// TIA Portal V20 export
// export: Created 2026-07-16T12:59:01.3797078Z, ExportSetting WithDefaults, DisplayName Totally Integrated Automation Portal, DisplayVersion V20 Update 5, DisplayName TIA Portal Openness, DisplayVersion V20 Update 4, DisplayName TIA Portal Version Control Interface, DisplayVersion V20 Update 5, DisplayName SINAMICS Startdrive Advanced, DisplayVersion V20, DisplayName SINAMICS DCC, DisplayVersion V20, DisplayName SINAMICS Startdrive G130, G150, S120, S150, SINAMICS MV, G220, S200, S210, DisplayVersion V20, DisplayName SINAMICS Startdrive G110M, G120, G120C, G120D, G120P, G115D, DisplayVersion V20, DisplayName STEP 7 Professional, DisplayVersion V20 Update 5, DisplayName STEP 7 Safety, DisplayVersion V20 Update 2, DisplayName WinCC Basic/Comfort/Advanced, DisplayVersion V20 Update 5, DisplayName WinCC Unified, DisplayVersion V20 Update 5
FUNCTION_BLOCK "FB_MotorFwdRevSystem"   // FB7, LAD
{ S7_Optimized_Access := 'TRUE' }
VERSION : 0.1
// stored: AutoNumber true, IsIECCheckEnabled false, IsRetainMemResEnabled false, MemoryReserve 100, SetENOAutomatically false, UDAEnableTagReadback false
   VAR RETAIN
      IO : "MotorFwdRevIOSet";
   END_VAR
   VAR
      RisingEdgeFlags : Array[0..3] of Bool;
      NegitiveSignalEdge : Array[0..2] of Bool;
      Pasue : Bool;
      HrTotaliserTimerReset : Bool;
      EnableUPSTimeMS : DInt;
      ShutdownTimeMS : DInt;
      FTTimeMS : DInt;
      PauseTimeMS : DInt;
      ReverseIgnoreFTTimeMS : DInt;
      FaultTripTimer { S7_SetPoint := 'True'} : TON_TIME;
      FTSTimer { S7_SetPoint := 'True'} : TON_TIME;
      EnableUpstreamTimer { S7_SetPoint := 'True'} : TON_TIME;
      ShutdownTimer { S7_SetPoint := 'True'} : TON_TIME;
      GeneralDelayTimer { S7_SetPoint := 'True'} : TON_TIME;
      InHandReqPreStart { S7_SetPoint := 'True'} : TON_TIME;
      CycleDelayReset { S7_SetPoint := 'True'} : TON_TIME;
   END_VAR
   VAR RETAIN
      HrTotaliserTimer { S7_SetPoint := 'True'} : TONR_TIME;
   END_VAR
   VAR
      ReversalPauseTimer { S7_SetPoint := 'True'} : TON_TIME;
      ReversalIgnoreFTTimer { S7_SetPoint := 'True'} : TON_TIME;
      PreStartMemory { S7_SetPoint := 'True'} : Bool;
      HandPosEdge : Bool;
      HandNegEdge : Bool;
      CycleDelay : Bool;
   END_VAR
   VAR_TEMP
      "Time" : Real;
      StartTimer : Bool;
   END_VAR
   VAR_TEMP   // added for the SCL form of the ladder/FBD networks
      _w1 : Bool;
      _w2 : Bool;
   END_VAR
BEGIN

REGION Network 1: Reverse Pause and Control
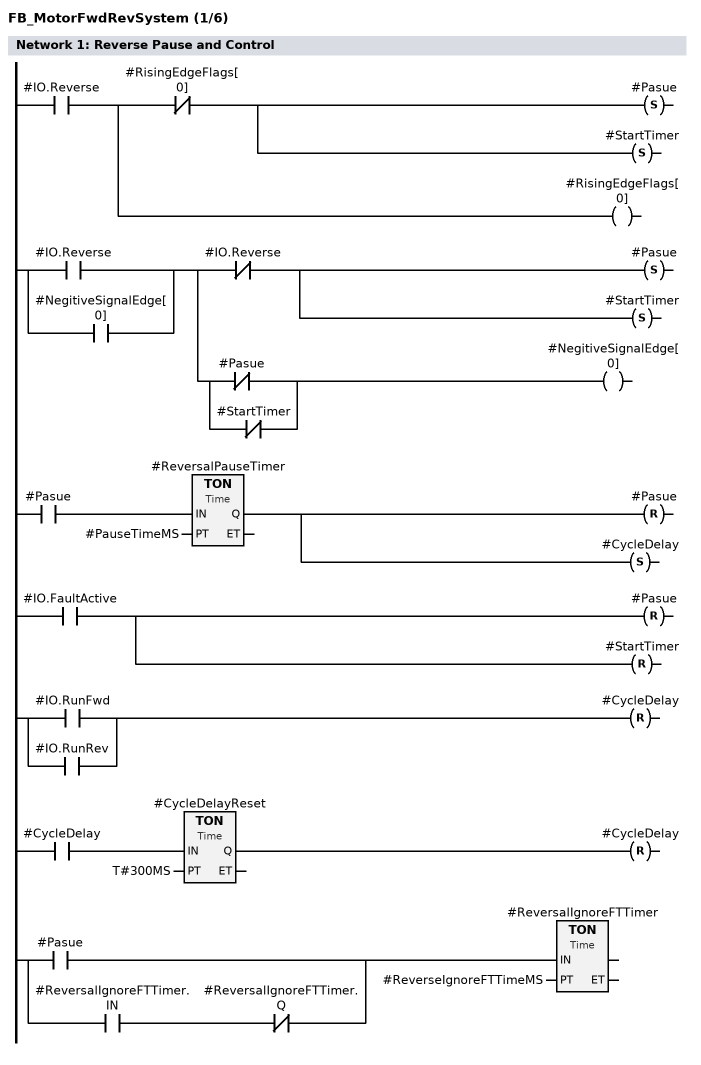
   RUNG wire#powerrail
      Contact( #IO.Reverse )
      wire#w1
      I_Contact( #RisingEdgeFlags[0] )
      wire#w2
      S_Coil( #Pasue )
   END_RUNG
   RUNG wire#w2
      S_Coil( #StartTimer )
   END_RUNG
   RUNG wire#w1
      Coil( #RisingEdgeFlags[0] )
   END_RUNG
   RUNG wire#powerrail
      Contact( #IO.Reverse )
      wire#w3
      I_Contact( #IO.Reverse )
      wire#w4
      S_Coil( #Pasue )
   END_RUNG
   RUNG wire#powerrail
      Contact( #NegitiveSignalEdge[0] )
   END_RUNG wire#w3
   RUNG wire#w4
      S_Coil( #StartTimer )
   END_RUNG
   RUNG wire#w3
      I_Contact( #Pasue )
      wire#w5
      Coil( #NegitiveSignalEdge[0] )
   END_RUNG
   RUNG wire#w3
      I_Contact( #StartTimer )
   END_RUNG wire#w5
   RUNG wire#powerrail
      Contact( #Pasue )
      { S7_Templates := "time_type := Time" } #ReversalPauseTimer.TON(pt := #PauseTimeMS, et =>)
      wire#w6
      R_Coil( #Pasue )
   END_RUNG
   RUNG wire#w6
      S_Coil( #CycleDelay )
   END_RUNG
   RUNG wire#powerrail
      Contact( #IO.FaultActive )
      wire#w7
      R_Coil( #Pasue )
   END_RUNG
   RUNG wire#w7
      R_Coil( #StartTimer )
   END_RUNG
   RUNG wire#powerrail
      Contact( #IO.RunFwd )
      wire#w8
      R_Coil( #CycleDelay )
   END_RUNG
   RUNG wire#powerrail
      Contact( #IO.RunRev )
   END_RUNG wire#w8
   RUNG wire#powerrail
      Contact( #CycleDelay )
      { S7_Templates := "time_type := Time" } #CycleDelayReset.TON(pt := T#300MS, et =>)
      R_Coil( #CycleDelay )
   END_RUNG
   RUNG wire#powerrail
      Contact( #Pasue )
      wire#w9
      { S7_Templates := "time_type := Time" } #ReversalIgnoreFTTimer.TON(pt := #ReverseIgnoreFTTimeMS, et =>)
   END_RUNG
   RUNG wire#powerrail
      Contact( #ReversalIgnoreFTTimer.IN )
      I_Contact( #ReversalIgnoreFTTimer.Q )
   END_RUNG wire#w9
   // the same network as SCL:
   IF #IO.Reverse AND NOT #RisingEdgeFlags[0] THEN
       #Pasue := TRUE;
       #StartTimer := TRUE;
   END_IF;
   #RisingEdgeFlags[0] := #IO.Reverse;
   #_w1 := #IO.Reverse OR #NegitiveSignalEdge[0];
   IF #_w1 AND NOT #IO.Reverse THEN
       #Pasue := TRUE;
       #StartTimer := TRUE;
   END_IF;
   #NegitiveSignalEdge[0] := #_w1 AND (NOT #Pasue OR NOT #StartTimer);
   #ReversalPauseTimer(IN := #Pasue, PT := #PauseTimeMS);   // TON
   IF #ReversalPauseTimer.Q THEN
       #Pasue := FALSE;
       #CycleDelay := TRUE;
   END_IF;
   IF #IO.FaultActive THEN
       #Pasue := FALSE;
       #StartTimer := FALSE;
   END_IF;
   IF #IO.RunFwd OR #IO.RunRev THEN #CycleDelay := FALSE; END_IF;
   #CycleDelayReset(IN := #CycleDelay, PT := T#300MS);   // TON
   IF #CycleDelayReset.Q THEN #CycleDelay := FALSE; END_IF;
   #ReversalIgnoreFTTimer(IN := #Pasue OR (#ReversalIgnoreFTTimer.IN AND NOT #ReversalIgnoreFTTimer.Q),   // TON
                          PT := #ReverseIgnoreFTTimeMS);
END_REGION

REGION Network 2: DOL Motor Start / Stop
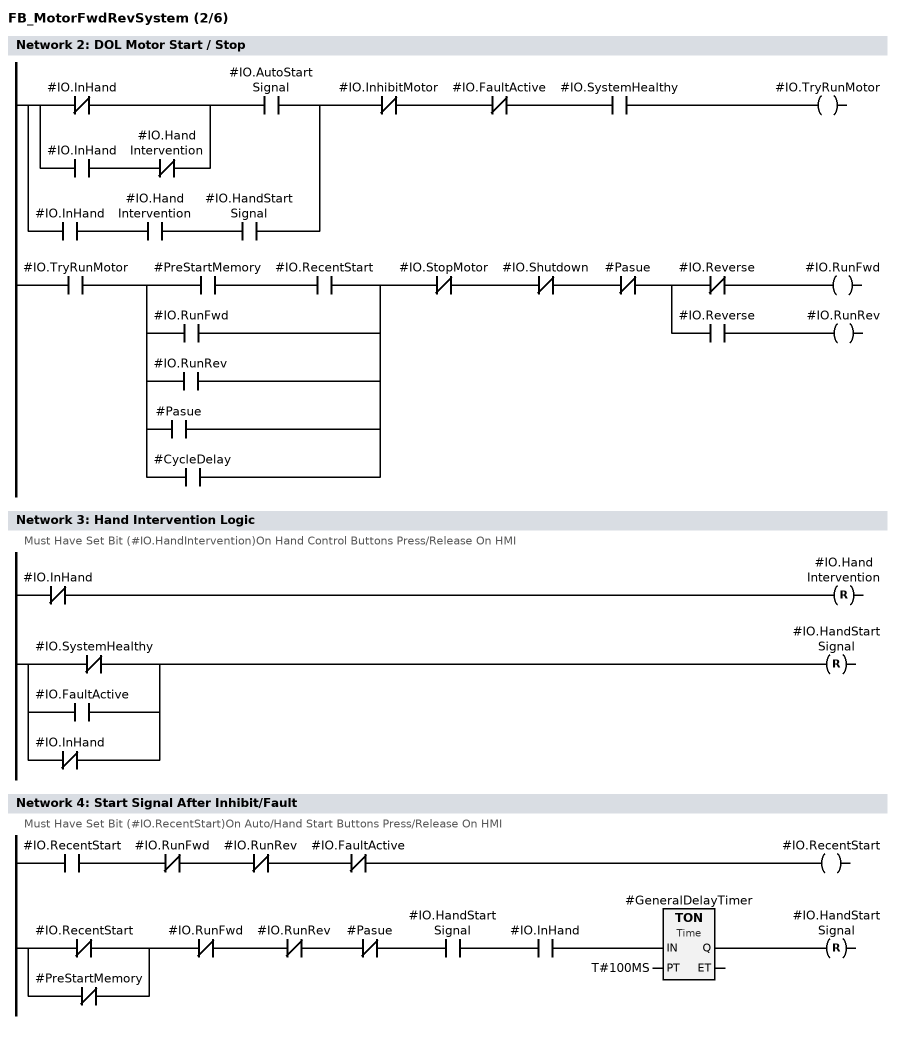
   RUNG wire#powerrail
      I_Contact( #IO.InHand )
      wire#w1
      Contact( #IO.AutoStartSignal )
      wire#w2
      I_Contact( #IO.InhibitMotor )
      I_Contact( #IO.FaultActive )
      Contact( #IO.SystemHealthy )
      Coil( #IO.TryRunMotor )
   END_RUNG
   RUNG wire#powerrail
      Contact( #IO.InHand )
      I_Contact( #IO.HandIntervention )
   END_RUNG wire#w1
   RUNG wire#powerrail
      Contact( #IO.InHand )
      Contact( #IO.HandIntervention )
      Contact( #IO.HandStartSignal )
   END_RUNG wire#w2
   RUNG wire#powerrail
      Contact( #IO.TryRunMotor )
      wire#w3
      Contact( #PreStartMemory )
      Contact( #IO.RecentStart )
      wire#w4
      I_Contact( #IO.StopMotor )
      I_Contact( #IO.Shutdown )
      I_Contact( #Pasue )
      wire#w5
      I_Contact( #IO.Reverse )
      Coil( #IO.RunFwd )
   END_RUNG
   RUNG wire#w3
      Contact( #IO.RunFwd )
   END_RUNG wire#w4
   RUNG wire#w3
      Contact( #IO.RunRev )
   END_RUNG wire#w4
   RUNG wire#w3
      Contact( #Pasue )
   END_RUNG wire#w4
   RUNG wire#w3
      Contact( #CycleDelay )
   END_RUNG wire#w4
   RUNG wire#w5
      Contact( #IO.Reverse )
      Coil( #IO.RunRev )
   END_RUNG
   // the same network as SCL:
   #IO.TryRunMotor := (((NOT #IO.InHand OR (#IO.InHand AND NOT #IO.HandIntervention)) AND #IO.AutoStartSignal) OR (#IO.InHand AND #IO.HandIntervention AND #IO.HandStartSignal)) AND NOT #IO.InhibitMotor AND NOT #IO.FaultActive AND #IO.SystemHealthy;
   #_w1 := #IO.TryRunMotor AND ((#PreStartMemory AND #IO.RecentStart) OR #IO.RunFwd OR #IO.RunRev OR #Pasue OR #CycleDelay) AND NOT #IO.StopMotor AND NOT #IO.Shutdown AND NOT #Pasue;
   #IO.RunFwd := #_w1 AND NOT #IO.Reverse;
   #IO.RunRev := #_w1 AND #IO.Reverse;
END_REGION

REGION Network 3: Hand Intervention Logic
   // Must Have Set Bit (#IO.HandIntervention)On Hand Control Buttons Press/Release On HMI
   RUNG wire#powerrail
      I_Contact( #IO.InHand )
      R_Coil( #IO.HandIntervention )
   END_RUNG
   RUNG wire#powerrail
      I_Contact( #IO.SystemHealthy )
      wire#w1
      R_Coil( #IO.HandStartSignal )
   END_RUNG
   RUNG wire#powerrail
      Contact( #IO.FaultActive )
   END_RUNG wire#w1
   RUNG wire#powerrail
      I_Contact( #IO.InHand )
   END_RUNG wire#w1
   // the same network as SCL:
   IF NOT #IO.InHand THEN #IO.HandIntervention := FALSE; END_IF;
   IF NOT #IO.SystemHealthy OR #IO.FaultActive OR NOT #IO.InHand THEN #IO.HandStartSignal := FALSE; END_IF;
END_REGION

REGION Network 4: Start Signal After Inhibit/Fault
   // Must Have Set Bit (#IO.RecentStart)On Auto/Hand Start Buttons Press/Release On HMI
   RUNG wire#powerrail
      Contact( #IO.RecentStart )
      I_Contact( #IO.RunFwd )
      I_Contact( #IO.RunRev )
      I_Contact( #IO.FaultActive )
      Coil( #IO.RecentStart )
   END_RUNG
   RUNG wire#powerrail
      I_Contact( #IO.RecentStart )
      wire#w1
      I_Contact( #IO.RunFwd )
      I_Contact( #IO.RunRev )
      I_Contact( #Pasue )
      Contact( #IO.HandStartSignal )
      Contact( #IO.InHand )
      { S7_Templates := "time_type := Time" } #GeneralDelayTimer.TON(pt := T#100MS, et =>)
      R_Coil( #IO.HandStartSignal )
   END_RUNG
   RUNG wire#powerrail
      I_Contact( #PreStartMemory )
   END_RUNG wire#w1
   // the same network as SCL:
   #IO.RecentStart := #IO.RecentStart AND NOT #IO.RunFwd AND NOT #IO.RunRev AND NOT #IO.FaultActive;
   #GeneralDelayTimer(IN := (NOT #IO.RecentStart OR NOT #PreStartMemory) AND NOT #IO.RunFwd AND NOT #IO.RunRev AND NOT #Pasue AND #IO.HandStartSignal AND #IO.InHand,   // TON
                      PT := T#100MS);
   IF #GeneralDelayTimer.Q THEN #IO.HandStartSignal := FALSE; END_IF;
END_REGION

REGION Network 5
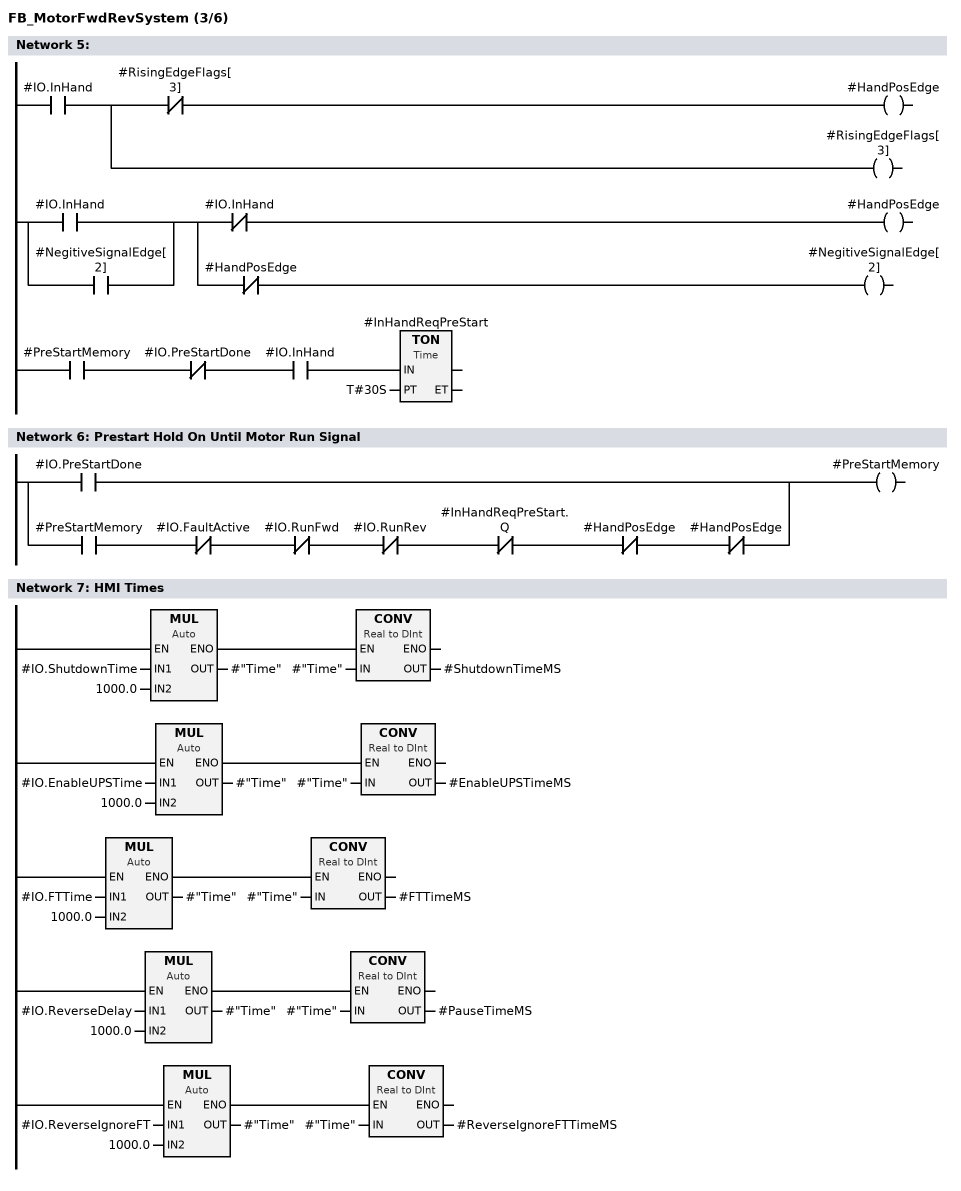
   RUNG wire#powerrail
      Contact( #IO.InHand )
      wire#w1
      I_Contact( #RisingEdgeFlags[3] )
      Coil( #HandPosEdge )
   END_RUNG
   RUNG wire#w1
      Coil( #RisingEdgeFlags[3] )
   END_RUNG
   RUNG wire#powerrail
      Contact( #IO.InHand )
      wire#w2
      I_Contact( #IO.InHand )
      Coil( #HandPosEdge )
   END_RUNG
   RUNG wire#powerrail
      Contact( #NegitiveSignalEdge[2] )
   END_RUNG wire#w2
   RUNG wire#w2
      I_Contact( #HandPosEdge )
      Coil( #NegitiveSignalEdge[2] )
   END_RUNG
   RUNG wire#powerrail
      Contact( #PreStartMemory )
      I_Contact( #IO.PreStartDone )
      Contact( #IO.InHand )
      { S7_Templates := "time_type := Time" } #InHandReqPreStart.TON(pt := T#30S, et =>)
   END_RUNG
   // the same network as SCL:
   #HandPosEdge := #IO.InHand AND NOT #RisingEdgeFlags[3];
   #RisingEdgeFlags[3] := #IO.InHand;
   #_w1 := #IO.InHand OR #NegitiveSignalEdge[2];
   #HandPosEdge := #_w1 AND NOT #IO.InHand;
   #NegitiveSignalEdge[2] := #_w1 AND NOT #HandPosEdge;
   #InHandReqPreStart(IN := #PreStartMemory AND NOT #IO.PreStartDone AND #IO.InHand, PT := T#30S);   // TON
END_REGION

REGION Network 6: Prestart Hold On Until Motor Run Signal
   RUNG wire#powerrail
      Contact( #IO.PreStartDone )
      wire#w1
      Coil( #PreStartMemory )
   END_RUNG
   RUNG wire#powerrail
      Contact( #PreStartMemory )
      I_Contact( #IO.FaultActive )
      I_Contact( #IO.RunFwd )
      I_Contact( #IO.RunRev )
      I_Contact( #InHandReqPreStart.Q )
      I_Contact( #HandPosEdge )
      I_Contact( #HandPosEdge )
   END_RUNG wire#w1
   // the same network as SCL:
   #PreStartMemory := #IO.PreStartDone OR (#PreStartMemory AND NOT #IO.FaultActive AND NOT #IO.RunFwd AND NOT #IO.RunRev AND NOT #InHandReqPreStart.Q AND NOT #HandPosEdge AND NOT #HandPosEdge);
END_REGION

REGION Network 7: HMI Times
   RUNG wire#powerrail
      Mul(in1 := #IO.ShutdownTime, in2 := 1000.0, out => #"Time")
      { S7_Templates := "[SrcType := Real, DestType := DInt]" } Convert(in := #"Time", out => #ShutdownTimeMS)
   END_RUNG
   RUNG wire#powerrail
      Mul(in1 := #IO.EnableUPSTime, in2 := 1000.0, out => #"Time")
      { S7_Templates := "[SrcType := Real, DestType := DInt]" } Convert(in := #"Time", out => #EnableUPSTimeMS)
   END_RUNG
   RUNG wire#powerrail
      Mul(in1 := #IO.FTTime, in2 := 1000.0, out => #"Time")
      { S7_Templates := "[SrcType := Real, DestType := DInt]" } Convert(in := #"Time", out => #FTTimeMS)
   END_RUNG
   RUNG wire#powerrail
      Mul(in1 := #IO.ReverseDelay, in2 := 1000.0, out => #"Time")
      { S7_Templates := "[SrcType := Real, DestType := DInt]" } Convert(in := #"Time", out => #PauseTimeMS)
   END_RUNG
   RUNG wire#powerrail
      Mul(in1 := #IO.ReverseIgnoreFT, in2 := 1000.0, out => #"Time")
      { S7_Templates := "[SrcType := Real, DestType := DInt]" } Convert(in := #"Time", out => #ReverseIgnoreFTTimeMS)
   END_RUNG
   // the same network as SCL:
   #"Time" := #IO.ShutdownTime * 1000.0;
   #ShutdownTimeMS := REAL_TO_DINT(#"Time");
   #"Time" := #IO.EnableUPSTime * 1000.0;
   #EnableUPSTimeMS := REAL_TO_DINT(#"Time");
   #"Time" := #IO.FTTime * 1000.0;
   #FTTimeMS := REAL_TO_DINT(#"Time");
   #"Time" := #IO.ReverseDelay * 1000.0;
   #PauseTimeMS := REAL_TO_DINT(#"Time");
   #"Time" := #IO.ReverseIgnoreFT * 1000.0;
   #ReverseIgnoreFTTimeMS := REAL_TO_DINT(#"Time");
END_REGION

REGION Network 8: DOL Motor Shutdown
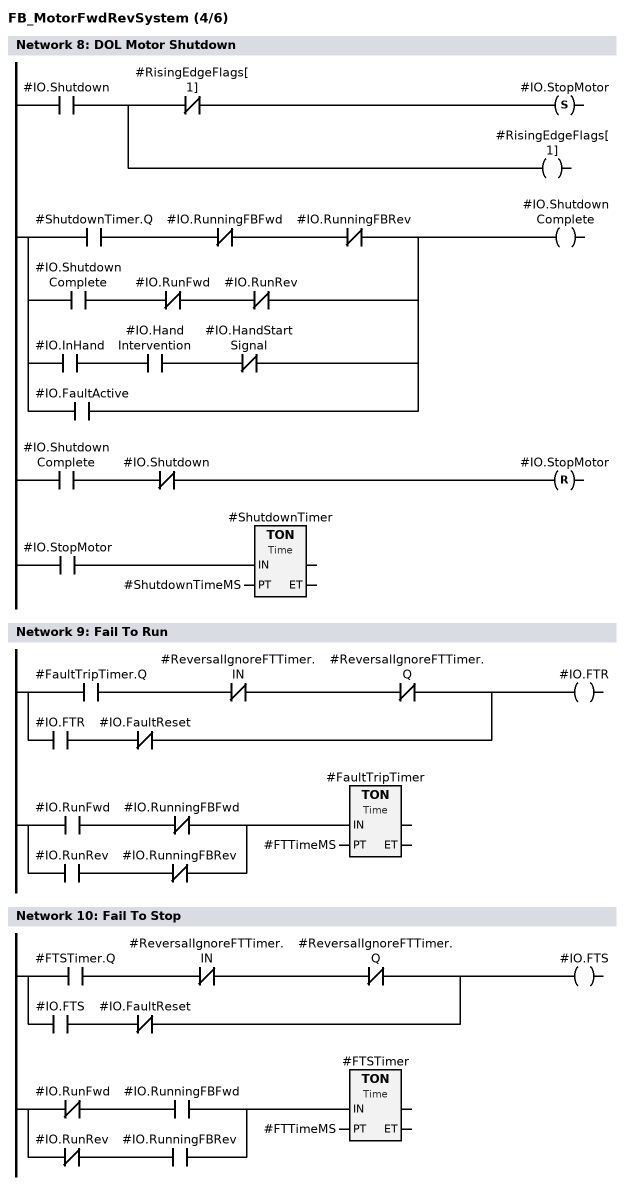
   RUNG wire#powerrail
      Contact( #IO.Shutdown )
      wire#w1
      I_Contact( #RisingEdgeFlags[1] )
      S_Coil( #IO.StopMotor )
   END_RUNG
   RUNG wire#w1
      Coil( #RisingEdgeFlags[1] )
   END_RUNG
   RUNG wire#powerrail
      Contact( #ShutdownTimer.Q )
      I_Contact( #IO.RunningFBFwd )
      I_Contact( #IO.RunningFBRev )
      wire#w2
      Coil( #IO.ShutdownComplete )
   END_RUNG
   RUNG wire#powerrail
      Contact( #IO.ShutdownComplete )
      I_Contact( #IO.RunFwd )
      I_Contact( #IO.RunRev )
   END_RUNG wire#w2
   RUNG wire#powerrail
      Contact( #IO.InHand )
      Contact( #IO.HandIntervention )
      I_Contact( #IO.HandStartSignal )
   END_RUNG wire#w2
   RUNG wire#powerrail
      Contact( #IO.FaultActive )
   END_RUNG wire#w2
   RUNG wire#powerrail
      Contact( #IO.ShutdownComplete )
      I_Contact( #IO.Shutdown )
      R_Coil( #IO.StopMotor )
   END_RUNG
   RUNG wire#powerrail
      Contact( #IO.StopMotor )
      { S7_Templates := "time_type := Time" } #ShutdownTimer.TON(pt := #ShutdownTimeMS, et =>)
   END_RUNG
   // the same network as SCL:
   IF #IO.Shutdown AND NOT #RisingEdgeFlags[1] THEN #IO.StopMotor := TRUE; END_IF;
   #RisingEdgeFlags[1] := #IO.Shutdown;
   #IO.ShutdownComplete := (#ShutdownTimer.Q AND NOT #IO.RunningFBFwd AND NOT #IO.RunningFBRev) OR (#IO.ShutdownComplete AND NOT #IO.RunFwd AND NOT #IO.RunRev) OR (#IO.InHand AND #IO.HandIntervention AND NOT #IO.HandStartSignal) OR #IO.FaultActive;
   IF #IO.ShutdownComplete AND NOT #IO.Shutdown THEN #IO.StopMotor := FALSE; END_IF;
   #ShutdownTimer(IN := #IO.StopMotor, PT := #ShutdownTimeMS);   // TON
END_REGION

REGION Network 9: Fail To Run
   RUNG wire#powerrail
      Contact( #FaultTripTimer.Q )
      I_Contact( #ReversalIgnoreFTTimer.IN )
      I_Contact( #ReversalIgnoreFTTimer.Q )
      wire#w1
      Coil( #IO.FTR )
   END_RUNG
   RUNG wire#powerrail
      Contact( #IO.FTR )
      I_Contact( #IO.FaultReset )
   END_RUNG wire#w1
   RUNG wire#powerrail
      Contact( #IO.RunFwd )
      I_Contact( #IO.RunningFBFwd )
      wire#w2
      { S7_Templates := "time_type := Time" } #FaultTripTimer.TON(pt := #FTTimeMS, et =>)
   END_RUNG
   RUNG wire#powerrail
      Contact( #IO.RunRev )
      I_Contact( #IO.RunningFBRev )
   END_RUNG wire#w2
   // the same network as SCL:
   #IO.FTR := (#FaultTripTimer.Q AND NOT #ReversalIgnoreFTTimer.IN AND NOT #ReversalIgnoreFTTimer.Q) OR (#IO.FTR AND NOT #IO.FaultReset);
   #FaultTripTimer(IN := (#IO.RunFwd AND NOT #IO.RunningFBFwd) OR (#IO.RunRev AND NOT #IO.RunningFBRev),   // TON
                   PT := #FTTimeMS);
END_REGION

REGION Network 10: Fail To Stop
   RUNG wire#powerrail
      Contact( #FTSTimer.Q )
      I_Contact( #ReversalIgnoreFTTimer.IN )
      I_Contact( #ReversalIgnoreFTTimer.Q )
      wire#w1
      Coil( #IO.FTS )
   END_RUNG
   RUNG wire#powerrail
      Contact( #IO.FTS )
      I_Contact( #IO.FaultReset )
   END_RUNG wire#w1
   RUNG wire#powerrail
      I_Contact( #IO.RunFwd )
      Contact( #IO.RunningFBFwd )
      wire#w2
      { S7_Templates := "time_type := Time" } #FTSTimer.TON(pt := #FTTimeMS, et =>)
   END_RUNG
   RUNG wire#powerrail
      I_Contact( #IO.RunRev )
      Contact( #IO.RunningFBRev )
   END_RUNG wire#w2
   // the same network as SCL:
   #IO.FTS := (#FTSTimer.Q AND NOT #ReversalIgnoreFTTimer.IN AND NOT #ReversalIgnoreFTTimer.Q) OR (#IO.FTS AND NOT #IO.FaultReset);
   #FTSTimer(IN := (NOT #IO.RunFwd AND #IO.RunningFBFwd) OR (NOT #IO.RunRev AND #IO.RunningFBRev),   // TON
             PT := #FTTimeMS);
END_REGION

REGION Network 11: Faults
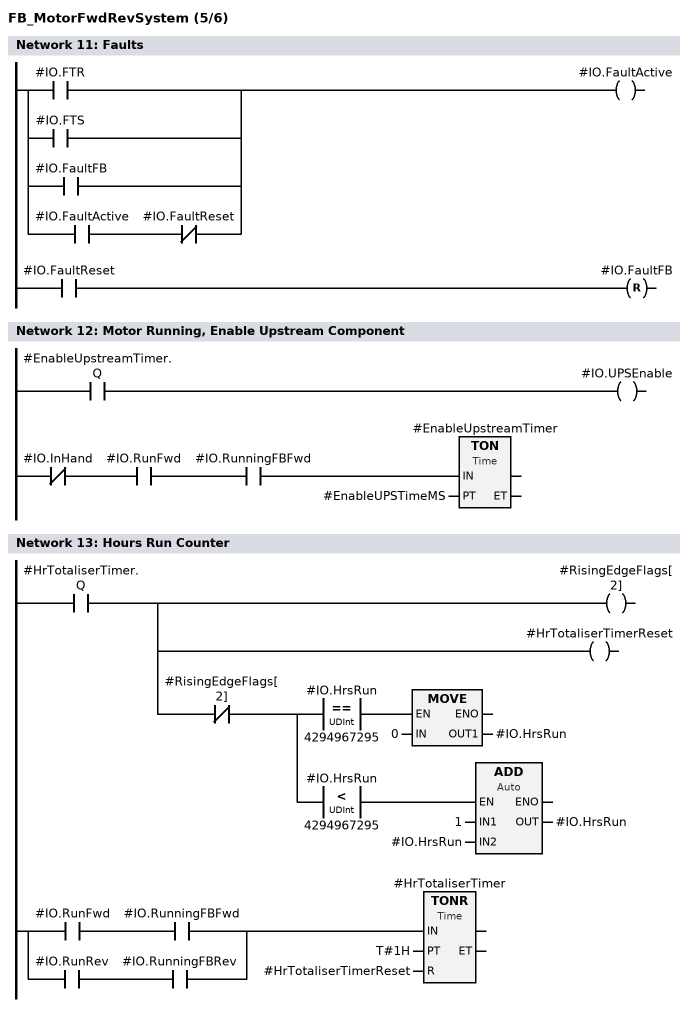
   RUNG wire#powerrail
      Contact( #IO.FTR )
      wire#w1
      Coil( #IO.FaultActive )
   END_RUNG
   RUNG wire#powerrail
      Contact( #IO.FTS )
   END_RUNG wire#w1
   RUNG wire#powerrail
      Contact( #IO.FaultFB )
   END_RUNG wire#w1
   RUNG wire#powerrail
      Contact( #IO.FaultActive )
      I_Contact( #IO.FaultReset )
   END_RUNG wire#w1
   RUNG wire#powerrail
      Contact( #IO.FaultReset )
      R_Coil( #IO.FaultFB )
   END_RUNG
   // the same network as SCL:
   #IO.FaultActive := #IO.FTR OR #IO.FTS OR #IO.FaultFB OR (#IO.FaultActive AND NOT #IO.FaultReset);
   IF #IO.FaultReset THEN #IO.FaultFB := FALSE; END_IF;
END_REGION

REGION Network 12: Motor Running, Enable Upstream Component
   RUNG wire#powerrail
      Contact( #EnableUpstreamTimer.Q )
      Coil( #IO.UPSEnable )
   END_RUNG
   RUNG wire#powerrail
      I_Contact( #IO.InHand )
      Contact( #IO.RunFwd )
      Contact( #IO.RunningFBFwd )
      { S7_Templates := "time_type := Time" } #EnableUpstreamTimer.TON(pt := #EnableUPSTimeMS, et =>)
   END_RUNG
   // the same network as SCL:
   #IO.UPSEnable := #EnableUpstreamTimer.Q;
   #EnableUpstreamTimer(IN := NOT #IO.InHand AND #IO.RunFwd AND #IO.RunningFBFwd, PT := #EnableUPSTimeMS);   // TON
END_REGION

REGION Network 13: Hours Run Counter
   RUNG wire#powerrail
      Contact( #HrTotaliserTimer.Q )
      wire#w1
      Coil( #RisingEdgeFlags[2] )
   END_RUNG
   RUNG wire#w1
      Coil( #HrTotaliserTimerReset )
   END_RUNG
   RUNG wire#w1
      I_Contact( #RisingEdgeFlags[2] )
      wire#w2
      { S7_Templates := "SrcType := UDInt" } EQ_Contact(in1 := #IO.HrsRun, in2 := 4294967295)
      Move(in := 0, out1 => #IO.HrsRun)
   END_RUNG
   RUNG wire#w2
      { S7_Templates := "SrcType := UDInt" } LT_Contact(in1 := #IO.HrsRun, in2 := 4294967295)
      Add(in1 := 1, in2 := #IO.HrsRun, out => #IO.HrsRun)
   END_RUNG
   RUNG wire#powerrail
      Contact( #IO.RunFwd )
      Contact( #IO.RunningFBFwd )
      wire#w3
      { S7_Templates := "time_type := Time" } #HrTotaliserTimer.TONR(pt := T#1H, et =>, r := #HrTotaliserTimerReset)
   END_RUNG
   RUNG wire#powerrail
      Contact( #IO.RunRev )
      Contact( #IO.RunningFBRev )
   END_RUNG wire#w3
   // the same network as SCL:
   #RisingEdgeFlags[2] := #HrTotaliserTimer.Q;
   #HrTotaliserTimerReset := #HrTotaliserTimer.Q;
   #_w1 := #HrTotaliserTimer.Q AND NOT #RisingEdgeFlags[2];
   IF #_w1 AND (#IO.HrsRun = 4294967295) THEN #IO.HrsRun := 0; END_IF;
   IF #_w1 AND (#IO.HrsRun < 4294967295) THEN #IO.HrsRun := 1 + #IO.HrsRun; END_IF;
   #HrTotaliserTimer(IN := (#IO.RunFwd AND #IO.RunningFBFwd) OR (#IO.RunRev AND #IO.RunningFBRev),   // TONR
                     PT := T#1H,
                     R := #HrTotaliserTimerReset);
END_REGION

REGION Network 14: HMI Motor Status Telemetry
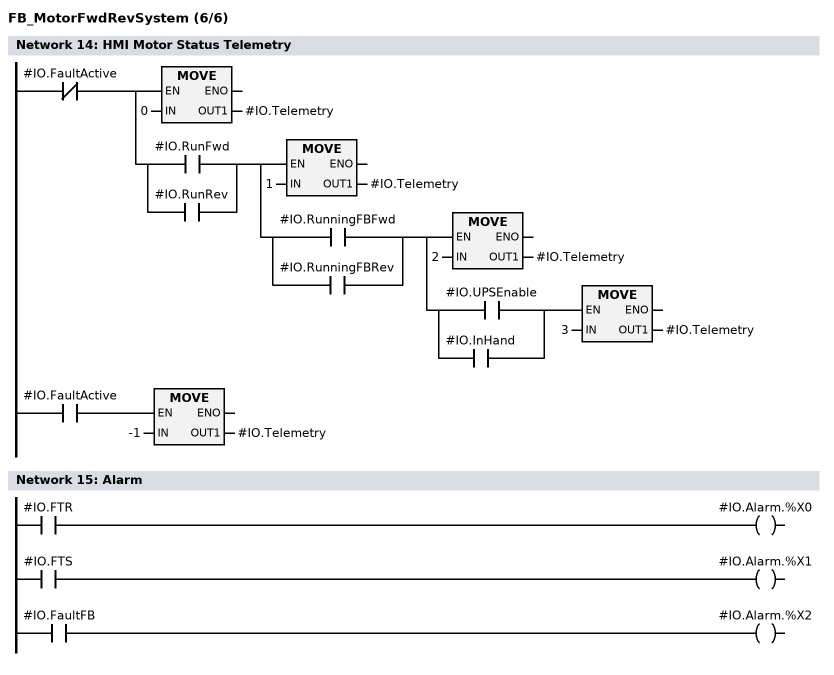
   RUNG wire#powerrail
      I_Contact( #IO.FaultActive )
      wire#w1
      Move(in := 0, out1 => #IO.Telemetry)
   END_RUNG
   RUNG wire#w1
      Contact( #IO.RunFwd )
      wire#w2
      Move(in := 1, out1 => #IO.Telemetry)
   END_RUNG
   RUNG wire#w1
      Contact( #IO.RunRev )
   END_RUNG wire#w2
   RUNG wire#w2
      Contact( #IO.RunningFBFwd )
      wire#w3
      Move(in := 2, out1 => #IO.Telemetry)
   END_RUNG
   RUNG wire#w2
      Contact( #IO.RunningFBRev )
   END_RUNG wire#w3
   RUNG wire#w3
      Contact( #IO.UPSEnable )
      wire#w4
      Move(in := 3, out1 => #IO.Telemetry)
   END_RUNG
   RUNG wire#w3
      Contact( #IO.InHand )
   END_RUNG wire#w4
   RUNG wire#powerrail
      Contact( #IO.FaultActive )
      Move(in := -1, out1 => #IO.Telemetry)
   END_RUNG
   // the same network as SCL:
   IF NOT #IO.FaultActive THEN #IO.Telemetry := 0; END_IF;
   #_w1 := NOT #IO.FaultActive AND (#IO.RunFwd OR #IO.RunRev);
   IF #_w1 THEN #IO.Telemetry := 1; END_IF;
   #_w2 := #_w1 AND (#IO.RunningFBFwd OR #IO.RunningFBRev);
   IF #_w2 THEN #IO.Telemetry := 2; END_IF;
   IF #_w2 AND (#IO.UPSEnable OR #IO.InHand) THEN #IO.Telemetry := 3; END_IF;
   IF #IO.FaultActive THEN #IO.Telemetry := -1; END_IF;
END_REGION

REGION Network 15: Alarm
   RUNG wire#powerrail
      Contact( #IO.FTR )
      Coil( #IO.Alarm.%X0 )
   END_RUNG
   RUNG wire#powerrail
      Contact( #IO.FTS )
      Coil( #IO.Alarm.%X1 )
   END_RUNG
   RUNG wire#powerrail
      Contact( #IO.FaultFB )
      Coil( #IO.Alarm.%X2 )
   END_RUNG
   // the same network as SCL:
   #IO.Alarm.%X0 := #IO.FTR;
   #IO.Alarm.%X1 := #IO.FTS;
   #IO.Alarm.%X2 := #IO.FaultFB;
END_REGION
END_FUNCTION_BLOCK
